// TIA Portal V19 export
TYPE "LEXCHANGETRAY_typePc_Cmd"
// stored: Access Published
   STRUCT
      simActive : Bool;
      execute : Bool;
      raiseError : Bool;
      resetError : Bool;
   END_STRUCT;
END_TYPE
